FUNCTION_BLOCK ALR2_SPLIT_FWD_REV (* ALR2 passthrough (Socket zu Plug) plus 2 ALR Plugs, die den Vorwaerts- und den Rueckwaerts-Kanal spiegeln *)
  (* Standard: 61499-2; Function: IN.EO1/DO1 (Vorwaerts, Indikation) wird unveraendert an OUT und zusaetzlich an FWD_OUT gespiegelt. OUT.EI1/DI1 (Rueckwaerts, Request) wird unveraendert an IN und zusaetzlich an REV_OUT gespiegelt.; Description: Copyright (c) 2026 HR Agrartechnik GmbH This program and the accompanying materials are made available under the terms of the Eclipse Public License 2.0 which is available at https://www.eclipse.org/legal/epl-2.0/ SPDX-License-Identifier: EPL-2.0 *)
  (* Version 1.0, 2026-09-21, Franz Höpfinger, HR Agrartechnik GmbH, Initial Version *)
  PACKAGE adapter::events::bidirectional;
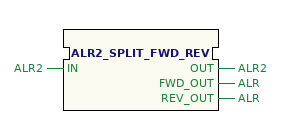
  SOCKETS
    IN : adapter::types::bidirectional::ALR2; (* bidirektionaler Eingang *)
  END_SOCKETS
  PLUGS
    OUT : adapter::types::bidirectional::ALR2; (* bidirektionaler Ausgang (Passthrough) *)
    FWD_OUT : adapter::types::unidirectional::ALR; (* spiegelt den Vorwaerts-Kanal (IN.EO1/DO1) *)
    REV_OUT : adapter::types::unidirectional::ALR; (* spiegelt den Rueckwaerts-Kanal (OUT.EI1/DI1) *)
  END_PLUGS
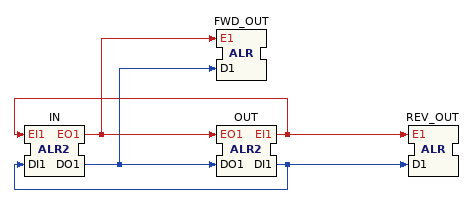
  EVENT_CONNECTIONS
    IN.EO1 TO OUT.EO1;
    IN.EO1 TO FWD_OUT.E1;
    OUT.EI1 TO IN.EI1;
    OUT.EI1 TO REV_OUT.E1;
  END_CONNECTIONS
  DATA_CONNECTIONS
    IN.DO1 TO OUT.DO1;
    IN.DO1 TO FWD_OUT.D1;
    OUT.DI1 TO IN.DI1;
    OUT.DI1 TO REV_OUT.D1;
  END_CONNECTIONS
END_FUNCTION_BLOCK
